(* IEC 61131-3 sources: Industry-PLC-LLM/data/PLCBEAD_repo/PLCBEAD_PLCEmbed-main/PLC-BEAD/Source/GEB/TEMP_NTC, 1 file *)

(* ---- TEMP_NTC.ST ---- *)
FUNCTION TEMP_NTC:REAL

VAR_INPUT
	RES :	REAL;
	RN :	REAL;
	B :	REAL;
END_VAR

IF RES > 0.0 THEN
	TEMP_NTC := B * 298.15 / (B + LN(RES / RN) * 298.15) -273.15;
END_IF;

END_FUNCTION

PROGRAM program0
  	VAR
		RES :	REAL;
		RN :	REAL;
		B :	REAL;
    	CEIL5_OUT : REAL;
  	END_VAR

  	CEIL5_OUT := TEMP_NTC(RES, RN, B);
END_PROGRAM
